
// ===== library types =====

FUNCTION_BLOCK "Tank"   // FB1, LAD
{ S7_Optimized_Access := 'TRUE' }
VERSION : 0.1
   VAR
      Level : Int;
      Tem : Int;
      Pre : Int;
   END_VAR
BEGIN
END_FUNCTION_BLOCK

(* ===== HMI "HMI_RT_1" =====

screen "根画面" 800x420
   Bar "棒图_1" at 46,14 size 80x230; MinimumValue 0; MaximumValue 100
*)

(* ===== HMI "HMI_RT_1" =====

screen "工厂" 800x420
   SymbolLibrary "符号库_1" at 153,31 size 536x285
*)

(* ===== HMI "HMI_RT_1" =====
system functions are stored by id; their names below are inferred from use
connection "HMI_连接_2": ETHERNET, S7_1500_OMS

HMI tags "默认变量表"
   "Tag_ScreenNumber" : UInt, internal

Template "Template_1" 800x420
   Button "退出" at 720,360 size 78x58; TextOn '退出 / Exit'; TextOff '退出 / Exit'; PictureOn "ExitRuntime_TP700_Comfort_TR"; PictureOff "ExitRuntime_TP700_Comfort_TR"
      on Release: StopRuntime(0)
   Button "Template_Button" at 640,360 size 78x58; TextOff 'Text'
   Button "Template_Button_1" at 560,360 size 78x58; TextOff 'Text'
   Button "Template_Button_2" at 480,360 size 78x58; TextOff 'Text'
   Button "Template_Button_3" at 400,360 size 78x58; TextOff 'Text'
   Button "Template_Button_4" at 321,360 size 78x58; TextOff 'Text'
   Button "Template_Button_5" at 241,360 size 78x58; TextOff 'Text'
   Button "Template_Button_6" at 161,360 size 78x58; TextOff 'Text'
   Button "报警" at 81,360 size 78x58; TextOn '报警 / Alarms'; TextOff '报警 / Alarms'; PictureOn "AlarmDisplay_TP700_Comfort_TR"; PictureOff "AlarmDisplay_TP700_Comfort_TR"
      on Release: function_ef3f5d25("报警窗口_Unacknowledged", -1)
   Button "起始画面" at 1,360 size 78x58; TextOn '起始画面 / Start screen'; TextOff '起始画面 / Start screen'; PictureOn "NavigateHome_TP700_Comfort_TR"; PictureOff "NavigateHome_TP700_Comfort_TR"
      on Release: ActivateScreen("Workshop1_DB", 0)
*)

(* ===== HMI "HMI_RT_1" =====

screen "IDB_车间2" 800x420
   TextField "文本域_1" at 551,78 size 41x20; Text 'Text'
*)

(* ===== HMI "HMI_RT_1" =====
system functions are stored by id; their names below are inferred from use

screen "根画面" 800x420, template "Template_1"
   on GenerateScreen: SetTag("Tag_ScreenNumber", 1)
   Button "按钮_1" at 2,2 size 96x32; TextOff '返回'
      on Click: ActivateScreen("工厂", 0)
*)

(* ===== HMI "HMI_RT_1" =====

screen "工厂" 800x420
   Button "Workshop1_DB_1" at 17,84 size 96x32; HelpText 'Workshop1_DB'; TextOff 'Text'
*)